FUNCTION_BLOCK C_HTTP_VERSION
VAR_INPUT
END_VAR
VAR_OUTPUT
END_VAR
VAR
	_Major : UINT := 1;
	_Minor : UINT := 0;
END_VAR

METHOD FB_init : BOOL
VAR_INPUT
	bInitRetains : BOOL; // if TRUE, the retain variables are initialized (warm start / cold start)
	bInCopyCode : BOOL;  // if TRUE, the instance afterwards gets moved into the copy code (online change)
	Major_Version : UINT;
	Minor_Version : UINT;
END_VAR
Major := Major_Version;
Minor := Minor_Version;
END_METHOD

PROPERTY Major : uint
GET
Major := _Major;
END_GET
SET
_Major := Major;
END_SET
END_PROPERTY

PROPERTY Minor : uint
GET
Minor := _Minor;
END_GET
SET
_Minor := Minor;
END_SET
END_PROPERTY

(*
	Y :		M:		D:
*)
METHOD Parse : RETURN_CODE
VAR_INPUT
	//String with format 'HTML/x.x'
		IN_STRING : STRING(255);
END_VAR
VAR
	_Fragment 		: STRING(255);
	_SubFragment 	: STRING(255);
	_i 				: INT;
END_VAR
_i := FIND(IN_STRING, '/');
IF _i = 0 THEN
	Parse := ph_lv0.LV0_RETURNCODE.RETURN_ERROR;
ELSE
	_Fragment := F_ToUCase(_Fragment);
	_Fragment := RIGHT(IN_STRING, LEN(IN_STRING) - _i);
	_i := FIND(_Fragment, '.');
	IF _i = 0 THEN
		Parse := ph_lv0.LV0_RETURNCODE.RETURN_ERROR;
	ELSE
		_SubFragment := RIGHT(_FRAGMENT, LEN(_FRAGMENT) - _i);
		_Fragment := LEFT(_FRAGMENT, _i - 1);
		Major := STRING_TO_UINT(_FRAGMENT);
		Minor := STRING_TO_UINT(_SubFragment);
		Parse := ph_lv0.LV0_RETURNCODE.RETURN_SUCCESS;
	END_IF
END_IF
END_METHOD

METHOD ToString : String(255)
VAR_INPUT
END_VAR
VAR
	_head 	: STRING(5) := 'HTML/';
END_VAR
ToString := CONCAT(_head, CONCAT(UINT_TO_STRING(_Major), CONCAT('.',UINT_TO_STRING(_Minor))));
END_METHOD

END_FUNCTION_BLOCK

(* stored: Version 1.1.0.1, ProductVersion 3.1.4019.2
   POU C_HTTP_VERSION: Id {f84bd680-1ef6-48ad-b83c-ad141d3ed4e4}, SpecialFunc None
   Method FB_init: Id {c34adc51-ee09-4037-b9e3-e4f48daea1dd}
   Property Major: Id {4b3fdcf0-e75c-4024-9e78-be75f2091c1e}
   Get Get: Id {ada1b26a-df10-46b8-8f9e-da84dce5f37a}
   Set Set: Id {b6631c3e-e518-4bd4-9b3e-5412be468414}
   Property Minor: Id {57502e27-2b87-4f07-b621-01f773a33730}
   Get Get: Id {e07d06e8-548f-488c-8910-2e3de44228c4}
   Set Set: Id {5e716222-489c-471d-b81a-506b30d80786}
   Method Parse: Id {f70f4b63-b7aa-461f-9c0f-ee6dd25eec59}
   Method ToString: Id {3fb1ece0-cd07-4895-a40e-68d34fc17c52} *)
